TYPE VTD_Motor_DUT :
STRUCT
	Enable:  BOOL;
	Enabled:  BOOL;
	Ready:  Bool;
	Running:  Bool;
	Forward:  Bool;
	Reverse:  Bool;
	Brake_Opened:  Bool;
	Speed:  Int;
	Speed_Actual:  Int;
	Actual_Current:  Int;
	Actual_Torque:  UInt;
	Acc_Factor:  UInt;
	Config_Axis:  Word;
	Error:  Bool;
	Status:  Word;
	Communication_Error:  Word;
	Lockout:  BOOL;
END_STRUCT
END_TYPE

(* stored: Version 1.1.0.1
   DUT VTD_Motor_DUT: Id {edbab4b6-9622-4d63-8741-16713e844ffb} *)
